ABB RobotStudio station: Trabalho Final_20220622-215942.rsstn

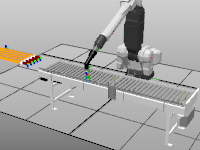
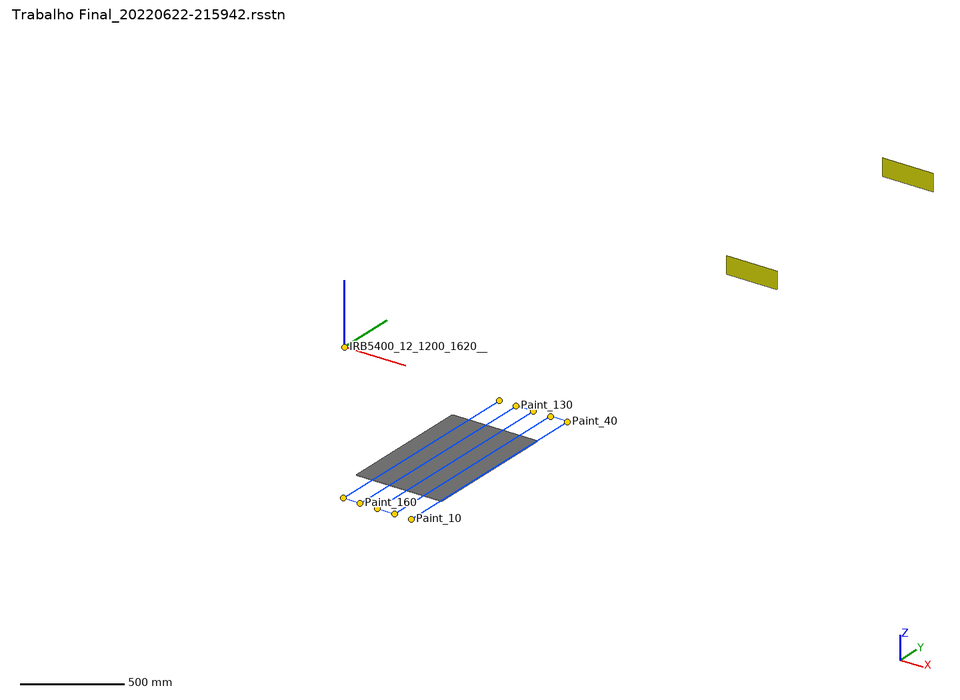
[picture v1: parts stored in the station drawn from their meshes, with robot base, taught points and paths (robot models come from the ABB library and are not in the file)]
Station Trabalho Final (saved by RobotStudio 21.4.9700.0)
Controller Controller_Pintura
  mechanical unit ROB_1: IRB5400_12_1200_1620__02, 6 joints, base frame (0, 0, 0) mm
Layout (positions relative to the parent item):
  - IRB5400_12_1200_1620__02 [mechanism, from Robots\IRB5400_12_1200_1620_G_02.rslib] at (0, 0, 0) mm; joint values [-0.0235, 0.1091, 0.4435, 1.7801, 0.0719, -1.7906] (rad or m)
  - ROBOBEL926_T_TD_03 [mechanism, from Tools\ROBOBEL926_T_TD_03.rslib] at (1967.84, -43.45, 1315.18) mm, rotated rx 180 ry 60 rz 179.94 deg
  - 600_guide [part, from Equipment\Conveyor Guide 600.rslib] at (1788.43, 1872.85, 0) mm, rotated rx 0 ry 0 rz -90.89 deg
  - Chapa [graphiccomponentgroup] at (0, -2160, 0) mm
    - Chapa_ParteDeCima [part] at (1817.02, -338.12, 823.77) mm, size 500 x 800 x 0 mm
    - Chapa_2 [part] at (1817.02, -338.12, 823.77) mm, size 500 x 800 x 0 mm
    - Chapa_3 [part] at (1817.02, -338.12, 823.77) mm, size 500 x 0 x 5 mm
    - Chapa_4 [part] at (1817.02, -338.12, 823.77) mm, size 0 x 800 x 5 mm
    - Chapa_5 [part] at (1817.02, -338.12, 823.77) mm, size 500 x 0 x 5 mm
    - Chapa_6 [part] at (1817.02, -338.12, 823.77) mm, size 0 x 800 x 5 mm
  - MeshModel_BoundingBox [graphiccomponentgroup]
  - MeshModel_ClippingPlane [graphiccomponentgroup]
  - MeshModel_ClippingCurve [graphiccomponentgroup]
  - SC_SprayFans [graphiccomponentgroup]
  - Positioner_2 [smart component, from Components\Positioner.rslib]
      properties: Object=Chapa; Position=[0 -2.16 0]; Orientation=[0 0 0]; Reference=Global; ReferenceObject=(none)
  - LinearMover_2 [smart component, from Components\LinearMover.rslib]
      properties: Object=Chapa; Direction=[0 1 0]; Speed=0.5; Reference=Global; ReferenceObject=(none)
  - PlaneSensor [smart component, from Components\PlaneSensor.rslib] at (1949.14, 396.86, 775.88) mm
      properties: Origin=[0 0 0]; Axis1=[0.3 0 0]; Axis2=[0 0 0.1]; SensedPart=(none)
    - _sensorPart_ [part], size 300 x 0 x 100 mm
  - LogicSRLatch [smart component, from Components\LogicSRLatch.rslib]
  - SimulationEvents [smart component, from Components\SimulationEvents.rslib]
  - PlaneSensor_2 [smart component, from Components\PlaneSensor.rslib] at (1949.14, 1699.17, 775.88) mm
      properties: Origin=[0 0 0]; Axis1=[0.3 0 0]; Axis2=[0 0 0.1]; SensedPart=(none)
    - _sensorPart_ [part], size 300 x 0 x 100 mm
Attachment: ROBOBEL926_T_TD_03 is attached to IRB5400_12_1200_1620__02 / Link6
Attachment: Workobject_Chapa is attached to Chapa
Station signals: DI Digital1
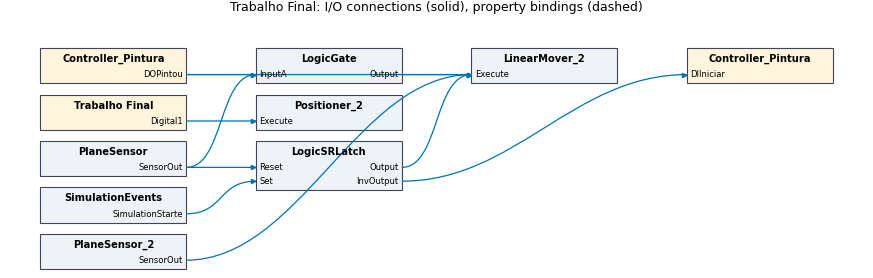
Station logic (signal -> signal, property => property):
  Controller_Pintura.DOPintou -> LogicGate.InputA
  Trabalho Final.Digital1 -> Positioner_2.Execute
  PlaneSensor.SensorOut -> LogicGate_2.InputA
  LogicGate_2.Output -> LinearMover_2.Execute
  PlaneSensor.SensorOut -> LogicSRLatch.Reset
  SimulationEvents.SimulationStarted -> LogicSRLatch.Set
  LogicSRLatch.Output -> LinearMover_2.Execute
  LogicSRLatch.InvOutput -> Controller_Pintura.DIIniciar
  Controller_Pintura.DOPintou -> LinearMover_2.Execute
  PlaneSensor_2.SensorOut -> LinearMover_2.Execute
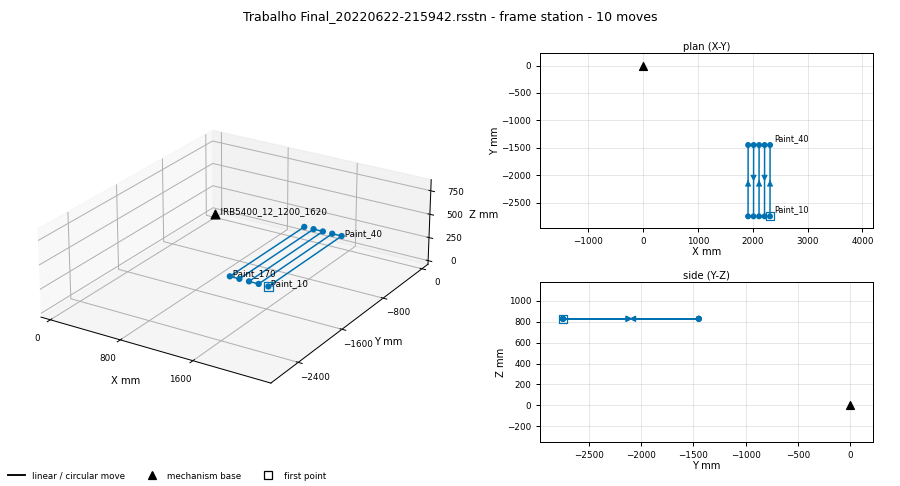
[picture p0: tool path of Trabalho Final_20220622-215942.rsstn in frame station, 10 of 10 moves have a stored position in this frame; points joined in program order, loops and branches not executed]
Targets, tools, work objects and paths stored in the station, written as RAPID:
! task (no controller)
MODULE BASE
  TASK PERS wobjdata Chapa_Parte_Superior:=[FALSE,TRUE,"",[[1817.023,-338.123,828.769],[1,0,0,0]],[[0,0,0],[1,0,0,0]]];
ENDMODULE

! task T_ROB1
MODULE CalibData
  PERS tooldata ROBOBEL926_T_TD_0:=[TRUE,[[117,0,470],[0.866025404,0,0.5,0]],[5.5,[30,0,225],[1,0,0,0],0,0,0]];
  PERS tooldata ROBOBEL926_T_TD_100:=[TRUE,[[204,0,520],[0.866025404,0,0.5,0]],[5.5,[30,0,225],[1,0,0,0],0,0,0]];
  PERS tooldata ROBOBEL926_T_TD_120:=[TRUE,[[220,0,530],[0.866025404,0,0.5,0]],[5.5,[30,0,225],[1,0,0,0],0,0,0]];
  PERS tooldata ROBOBEL926_T_TD_150:=[TRUE,[[247,0,545],[0.866025404,0,0.5,0]],[5.5,[30,0,225],[1,0,0,0],0,0,0]];
  PERS tooldata ROBOBEL926_T_TD_200:=[TRUE,[[290,0,570],[0.866025404,0,0.5,0]],[5.5,[30,0,225],[1,0,0,0],0,0,0]];
  PERS tooldata ROBOBEL926_T_TD_250:=[TRUE,[[333,0,595],[0.866025404,0,0.5,0]],[5.5,[30,0,225],[1,0,0,0],0,0,0]];
  PERS tooldata ROBOBEL926_T_TD_300:=[TRUE,[[377,0,620],[0.866025404,0,0.5,0]],[5.5,[30,0,225],[1,0,0,0],0,0,0]];
ENDMODULE

! task T_ROB1
MODULE m4
  LOCAL CONST robtarget Paint_10:=[[498.743494875,-249.999639638,-0.000355856],[0,0.000512373,0.999999869,0],[-1,1,-2,0],[9E+09,9E+09,9E+09,9E+09,9E+09,9E+09]];
  LOCAL CONST robtarget Paint_40:=[[500.075664199,1050.000097836,-0.000355856],[0,0.000512373,0.999999869,0],[0,0,-1,0],[9E+09,9E+09,9E+09,9E+09,9E+09,9E+09]];
  LOCAL CONST robtarget Paint_50:=[[400.075559403,1050.000097836,-0.000355856],[0,0.000512373,0.999999869,0],[0,0,-1,0],[9E+09,9E+09,9E+09,9E+09,9E+09,9E+09]];
  LOCAL CONST robtarget Paint_80:=[[398.743390079,-249.999639638,-0.000355856],[0,0.000512373,0.999999869,0],[-1,1,-2,0],[9E+09,9E+09,9E+09,9E+09,9E+09,9E+09]];
  LOCAL CONST robtarget Paint_90:=[[298.743285283,-249.999639638,-0.000355856],[0,0.000512373,0.999999869,0],[-1,1,-2,0],[9E+09,9E+09,9E+09,9E+09,9E+09,9E+09]];
  LOCAL CONST robtarget Paint_120:=[[300.075454607,1050.000097836,-0.000355856],[0,0.000512373,0.999999869,0],[0,0,0,0],[9E+09,9E+09,9E+09,9E+09,9E+09,9E+09]];
  LOCAL CONST robtarget Paint_130:=[[200.075349811,1050.000097836,-0.000355856],[0,0.000512373,0.999999869,0],[0,0,0,0],[9E+09,9E+09,9E+09,9E+09,9E+09,9E+09]];
  LOCAL CONST robtarget Paint_160:=[[198.743180487,-249.999639638,-0.000355856],[0,0.000512373,0.999999869,0],[-1,1,-2,0],[9E+09,9E+09,9E+09,9E+09,9E+09,9E+09]];
  LOCAL CONST robtarget Paint_170:=[[98.743075691,-249.999639638,-0.000355856],[0,0.000512373,0.999999869,0],[-1,1,-2,0],[9E+09,9E+09,9E+09,9E+09,9E+09,9E+09]];
  LOCAL CONST robtarget Paint_200:=[[100.075245015,1050.000097836,-0.000355856],[0,0.000512373,0.999999869,0],[0,0,0,0],[9E+09,9E+09,9E+09,9E+09,9E+09,9E+09]];
  PROC mainm4()
  ENDPROC
  PROC Chapa_Panel_1()
    PaintL Paint_10,v800,z100,ROBOBEL926_T_TD_150\WObj:=Workobject_Chapa;
    SetBrush 3\Y:=-100;
    SetBrush 1\Y:=900;
    PaintL Paint_40,v800,z100,ROBOBEL926_T_TD_150\WObj:=Workobject_Chapa;
    PaintL Paint_50,v800,z100,ROBOBEL926_T_TD_150\WObj:=Workobject_Chapa;
    SetBrush 3\Y:=900;
    SetBrush 1\Y:=-100;
    PaintL Paint_80,v800,z100,ROBOBEL926_T_TD_150\WObj:=Workobject_Chapa;
    PaintL Paint_90,v800,z100,ROBOBEL926_T_TD_150\WObj:=Workobject_Chapa;
    SetBrush 3\Y:=-100;
    SetBrush 1\Y:=900;
    PaintL Paint_120,v800,z100,ROBOBEL926_T_TD_150\WObj:=Workobject_Chapa;
    PaintL Paint_130,v800,z100,ROBOBEL926_T_TD_150\WObj:=Workobject_Chapa;
    SetBrush 3\Y:=900;
    SetBrush 1\Y:=-100;
    PaintL Paint_160,v800,z100,ROBOBEL926_T_TD_150\WObj:=Workobject_Chapa;
    PaintL Paint_170,v800,z100,ROBOBEL926_T_TD_150\WObj:=Workobject_Chapa;
    SetBrush 3\Y:=-100;
    SetBrush 1\Y:=900;
    PaintL Paint_200,v800,z100,ROBOBEL926_T_TD_150\WObj:=Workobject_Chapa;
  ENDPROC
ENDMODULE

! task T_ROB1
MODULE BASE
  TASK PERS wobjdata Workobject_Chapa:=[FALSE,TRUE,"",[[1817.023,-2498.123,828.769],[1,0,0,0]],[[0,0,0],[1,0,0,0]]];
ENDMODULE

! task T_ROB1
MODULE pntexstart
  PROC ExStartReset()
  ENDPROC
  PROC WaitExStart()
    WaitTime 0.1;
  ENDPROC
ENDMODULE

! task T_ROB1
MODULE posmsg
  PROC PostMainPosMsg()
  ENDPROC
  PROC PreMainPosMsg()
  ENDPROC
ENDMODULE

! task T_ROB1
MODULE pntloop
  LOCAL VAR signaldo doJobCompAlias;
  PROC main()
    CallInitCustMain;
    ClearCurrentJob;
    Reset doJobCompAlias;
    PulseDO \High\PLength:=2.0,doJobCompAlias;
    ClearCurrentJob;
    WaitTime 0.2;
    Chapa_Panel_1;
  ENDPROC
  LOCAL PROC ClearCurrentJob()
  ENDPROC
  PROC CallInitCustMain()
  ENDPROC
ENDMODULE

! task T_ROB1
MODULE sysdata
  PROC PowerOnWZones()
  ENDPROC
  PROC ConfSettingsOff()
    ConfJ \Off;
    ConfL \Off;
  ENDPROC
ENDMODULE

! task T_ROB1
MODULE custmain
  PROC PreMainCustom()
  ENDPROC
  PROC InitCustMain()
  ENDPROC
  PROC PostMainCustom()
  ENDPROC
ENDMODULE

! task T_ROB1
MODULE pntprogmap
  PROC SetProgramModule()
  ENDPROC
ENDMODULE

! task T_ROB1
MODULE pnttipclean
  PROC TipCleanPreMain()
    AppCleanRun;
    TipCleanRun;
    TipCleanRun;
    AppCleanRun;
  ENDPROC
  PROC TipCleanPostMain()
    AppCleanRun;
    TipCleanRun;
    TipCleanRun;
    AppCleanRun;
  ENDPROC
  PROC TipCleanRun()
  ENDPROC
  PROC AppCleanRun()
  ENDPROC
ENDMODULE

